FUNCTION_BLOCK SafetyMonFB_TcEvents EXTENDS SafetyBase IMPLEMENTS I_EventReactionTcEvents, I_InSafetyGroup
VAR
	{attribute 'hide'}
	_ActiveAlarm : BOOL := TRUE;
	{attribute 'hide'}
	_ActiveName	 : STRING := 'pressed!';
	Events		 : TcEventClass('Safety MonFB Events');
	_SafetyGroup : I_TaskResult;
END_VAR

PROPERTY ActiveAlarm : BOOL
SET
_ActiveAlarm := ActiveAlarm;
END_SET
END_PROPERTY

PROPERTY ActiveName : STRING
SET
_ActiveName := ActiveName;
END_SET
END_PROPERTY

METHOD CyclicLogic
SUPER^.CyclicLogic();
_OK	   := SUPER^.InfoData.State = E_SafetyMon_State.Run;
_Error := GetHighestActiveEventReaction() >= TcEventSeverity.Error;
IF _SafetyGroup <> 0 THEN
	IF _SafetyGroup.Error THEN
		Events.Reset();
		RETURN;
	END_IF
END_IF

IF _ResetFunction <> 0 AND_THEN _ResetFunction.Busy THEN
	RETURN;
END_IF

IF NOT SUPER^.OK AND _ActiveAlarm THEN
	Events.Arguments(E_SafetyMon.Active).Clear().AddString(_ActiveName);
	Events.RaiseEvent(E_SafetyMon.Active);
END_IF

IF SUPER^.InfoData.Diag.0 THEN
	Events.RaiseEvent(E_SafetyMon.Disc1);
END_IF

IF SUPER^.InfoData.Diag.1 THEN
	Events.RaiseEvent(E_SafetyMon.Disc2);
END_IF

IF SUPER^.InfoData.Diag.2 THEN
	Events.RaiseEvent(E_SafetyMon.DiscInput);
END_IF

IF SUPER^.InfoData.Diag.4 THEN
	Events.RaiseEvent(E_SafetyMon.Edm1);
END_IF

IF SUPER^.InfoData.Diag.5 THEN
	Events.RaiseEvent(E_SafetyMon.Edm2);
END_IF

IF SUPER^.InfoData.Diag.8 THEN
	Events.RaiseEvent(E_SafetyMon.Disc1Safe);
END_IF

IF SUPER^.InfoData.Diag.9 THEN
	Events.RaiseEvent(E_SafetyMon.Disc2Safe);
END_IF

IF SUPER^.InfoData.Diag.10 THEN
	Events.RaiseEvent(E_SafetyMon.DiscInputSafe);
END_IF
END_METHOD

(*FB_Init is always available implicitly and it is used primarily for initialization.
The return value is not evaluated. For a specific influence, you can also declare the
methods explicitly and provide additional code there with the standard initialization
code. You can evaluate the return value.*)
METHOD FB_Init : BOOL
VAR_INPUT
	(* TRUE: the retain variables are initialized (reset warm / reset cold)*)
	bInitRetains : BOOL;

	(* TRUE: the instance will be copied to the copy code afterward (online change)   *)
	bInCopyCode : BOOL;
	Name		: T_MaxString;
END_VAR
Events.GenerateTcEvents(Name, ADR(TC_events.SafetyMon), SIZEOF(ST_SafetyMon));
END_METHOD

METHOD GetHighestActiveEventReaction : DINT
GetHighestActiveEventReaction := Events.GetHighestActiveEventReaction();
END_METHOD

METHOD GetHighestActiveEventSeverity : TcEventSeverity
GetHighestActiveEventSeverity := Events.GetHighestActiveEventSeverity();
END_METHOD

METHOD Reset
SUPER^.Reset();
Events.Reset();
END_METHOD

PROPERTY SafetyGroup : I_TaskResult
SET
_SafetyGroup := SafetyGroup;
END_SET
END_PROPERTY

METHOD SetEventReactions
VAR_INPUT
	Verbose	 : DINT := 0;
	Info	 : DINT := 1;
	Warning	 : DINT := 2;
	Error	 : DINT := 3;
	Critical : DINT := 4;
END_VAR
Events.SetEventReactions(Verbose,
						 Info,
						 Warning,
						 Error,
						 Critical);
END_METHOD

END_FUNCTION_BLOCK

(* stored: Version 1.1.0.1, ProductVersion 3.1.4026.18
   POU SafetyMonFB_TcEvents: Id {67adfd40-9596-4cff-9ae8-120b3bef74c1}, SpecialFunc None
   Folder Cyclic: Id {78c651f7-e687-4f22-bfc4-094037c59675}
   Folder Events: Id {146a2dd2-8c83-4226-9a84-8ac6e48836a8}
   Property ActiveAlarm: Id {5113c18b-ebe0-00f4-3202-4c1830b7105d}
   Set Set: Id {773800b8-ff2d-055f-1908-63b0aa36c0b5}
   Property ActiveName: Id {edba08d8-6c67-0382-2f69-477f60bcff69}
   Set Set: Id {a4917e4b-797e-0eeb-390a-59efcf21fb43}
   Method CyclicLogic: Id {65730a53-ecec-4366-ba15-e31222aa9cae}
   Method FB_Init: Id {fb7afd79-b20b-4503-ac65-cef031c9c063}
   Method GetHighestActiveEventReaction: Id {7c7c2702-eecf-4e0b-9c82-5bb8333599b9}
   Method GetHighestActiveEventSeverity: Id {7eafac5e-b51d-4382-bd58-4f520dbba2ee}
   Method Reset: Id {893ecc6b-83ee-4eff-a2d7-ab383932f614}
   Property SafetyGroup: Id {419ee011-d34a-495e-9034-1bb438cb9f42}
   Set Set: Id {4acfbcff-26c3-40aa-8574-2a08711f5cbb}
   Method SetEventReactions: Id {10bb5c42-2cc5-4bd0-977b-b09f2f24c084} *)
